(* IEC 61131-3 sources: ae-debugging/src, 4 files *)

(* ---- typeMotor.st ---- *)
TYPE
    Motor : STRUCT
        is_running        : BOOL    ;
        power_consumption : REAL    := 369;
        hours_operating   : INT     := 10;
    END_STRUCT;
END_TYPE

(* ---- class.st ---- *)
CLASS Conveyor
    VAR PRIVATE
        Motor1 : Motor;
        Motor2 : Motor;
    END_VAR

    VAR PUBLIC
        is_running : BOOL;
    END_VAR

    METHOD PUBLIC Start
        Motor1.is_running := TRUE;
        Motor2.is_running := TRUE;
        is_running := TRUE;
    END_METHOD

    METHOD PUBLIC Stop
        Motor1.is_running := FALSE;
        Motor2.is_running := FALSE;
        is_running := FALSE;
    END_METHOD
END_CLASS

(* ---- configuration.st ---- *)
CONFIGURATION PLC_1
    VAR_GLOBAL
        GlobalInt : int;
        UpCounterInt : int;
    END_VAR

    TASK Main1(Interval := T#300ms, Priority := 1);
        PROGRAM P1 WITH Main1 : FuncProgram;
        PROGRAM P2 WITH Main1 : ClassProgram;

    TASK Main2(Interval := T#10ms, Priority := 1);
        PROGRAM P3 WITH Main2 : FbProgram;
END_CONFIGURATION

(* ---- fbProgram.st ---- *)
PROGRAM FbProgram
    VAR_EXTERNAL
        UpCounterInt : int;
    END_VAR

    VAR
        functionBlock : fb;
    END_VAR

    UpCounterInt := UpCounterInt + 1;

    functionBlock();

END_PROGRAM
